FUNCTION_BLOCK CentralServerConveyorCTL (* Basic Function Block Type *)
  (* Standard: 61499-2 *)
  (* Version 0.2, 2003-12-04, JHC, Rockwell Automation, Renamed for better indexing. *)
  (* Version 0.1, 2002-11-05, JHC, Rockwell Automation, Corrected missing ST element in Algorithm REQ. *)
  (* Version 0.0, 2000-05-30, JHC, Rockwell Automation *)
  (* Compiler header: package fb.rt.cs725; *)
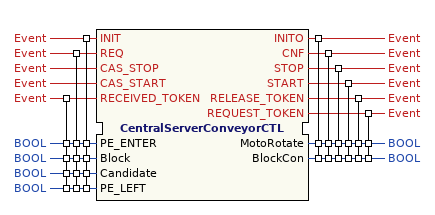
  EVENT_INPUT
    INIT WITH PE_ENTER, Block, Candidate, PE_LEFT; (* Initialization Request *)
    REQ WITH PE_ENTER, Block, Candidate, PE_LEFT; (* Normal Execution Request *)
    CAS_STOP;
    CAS_START;
    RECEIVED_TOKEN WITH PE_ENTER, Block, Candidate, PE_LEFT;
  END_EVENT
  EVENT_OUTPUT
    INITO WITH MotoRotate, BlockCon; (* Initialization Confirm *)
    CNF WITH MotoRotate, BlockCon; (* Execution Confirmation *)
    STOP WITH MotoRotate, BlockCon;
    START WITH BlockCon, MotoRotate;
    RELEASE_TOKEN WITH MotoRotate, BlockCon;
    REQUEST_TOKEN WITH MotoRotate, BlockCon;
  END_EVENT
  VAR_INPUT
    PE_ENTER : BOOL; (* Input event qualifier *)
    Block : BOOL;
    Candidate : BOOL;
    PE_LEFT : BOOL;
  END_VAR
  VAR_OUTPUT
    MotoRotate : BOOL; (* Output event qualifier *)
    BlockCon : BOOL;
  END_VAR
  VAR
    lastPE : BOOL := 1;
    lastBlock : BOOL := 0;
  END_VAR
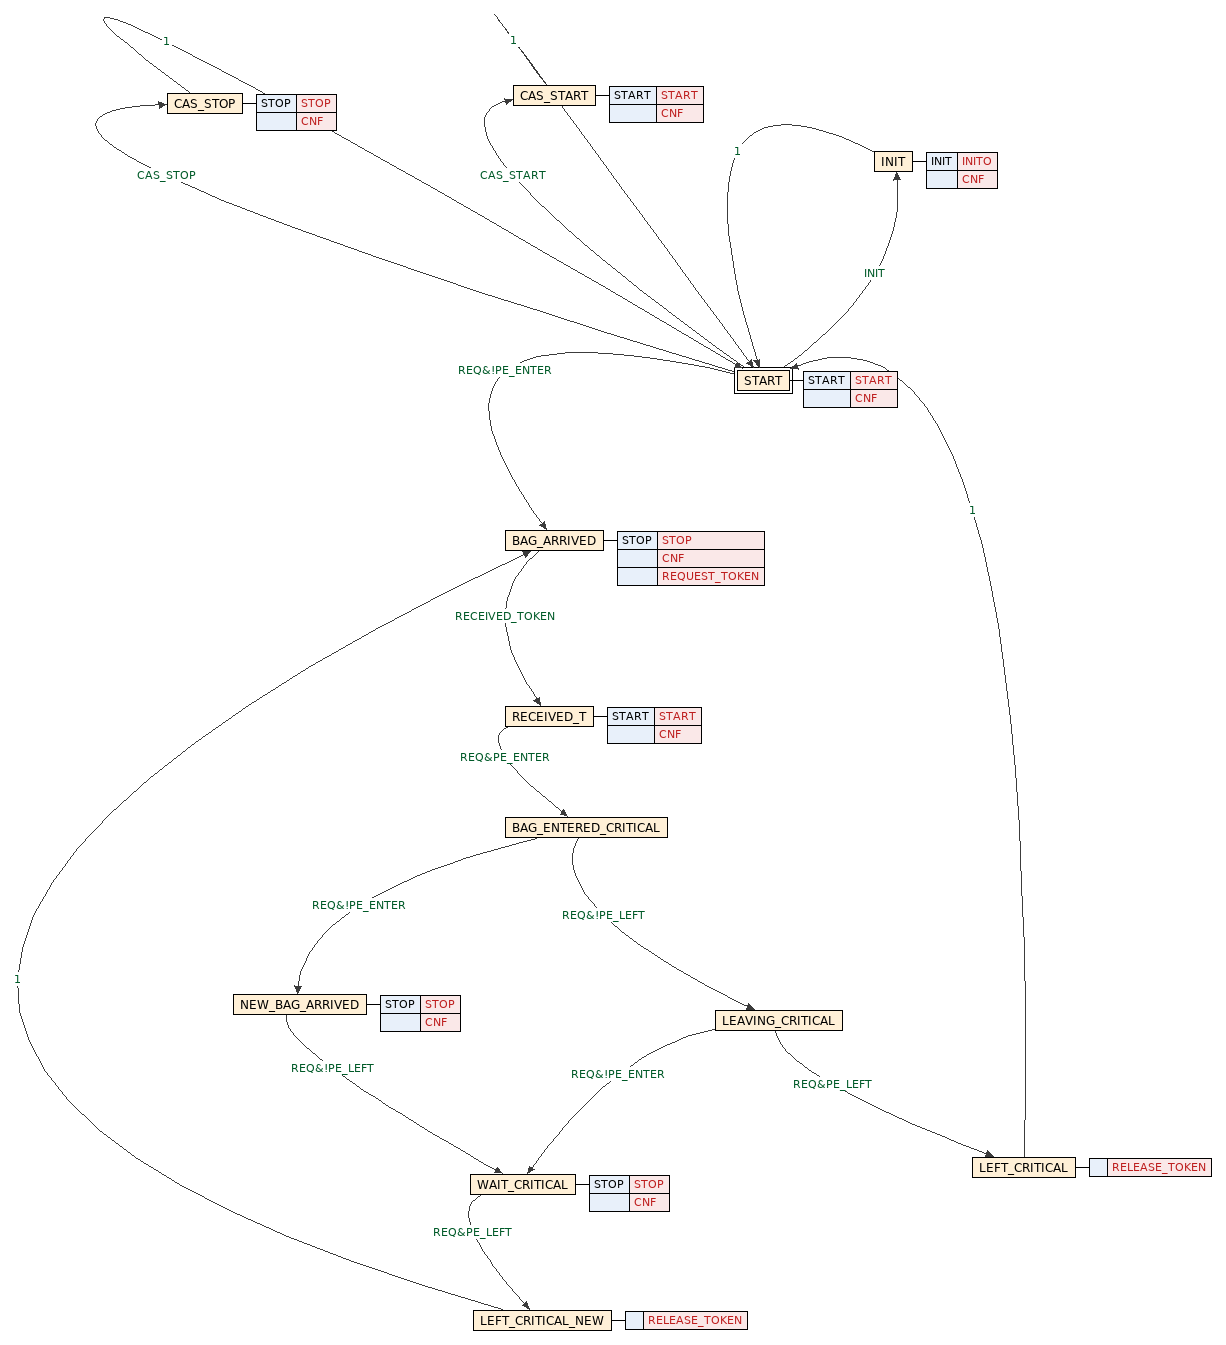
  EC_STATES
    START : START -> START, -> CNF; (* Initial State *)
    INIT : INIT -> INITO, -> CNF; (* Initialization *)
    BAG_ARRIVED : STOP -> STOP, -> CNF, -> REQUEST_TOKEN; (* Normal execution *)
    CAS_START : START -> START, -> CNF;
    CAS_STOP : STOP -> STOP, -> CNF;
    RECEIVED_T : START -> START, -> CNF; (* Token recived *)
    BAG_ENTERED_CRITICAL;
    NEW_BAG_ARRIVED : STOP -> STOP, -> CNF;
    LEAVING_CRITICAL;
    WAIT_CRITICAL : STOP -> STOP, -> CNF;
    LEFT_CRITICAL_NEW : -> RELEASE_TOKEN;
    LEFT_CRITICAL : -> RELEASE_TOKEN;
  END_STATES
  EC_TRANSITIONS
    START TO INIT := INIT;
    INIT TO START := 1;
    START TO BAG_ARRIVED := REQ&!PE_ENTER;
    START TO CAS_START := CAS_START;
    CAS_START TO START := 1;
    START TO CAS_STOP := CAS_STOP;
    CAS_STOP TO START := 1;
    BAG_ARRIVED TO RECEIVED_T := RECEIVED_TOKEN;
    RECEIVED_T TO BAG_ENTERED_CRITICAL := REQ&PE_ENTER;
    BAG_ENTERED_CRITICAL TO NEW_BAG_ARRIVED := REQ&!PE_ENTER;
    BAG_ENTERED_CRITICAL TO LEAVING_CRITICAL := REQ&!PE_LEFT;
    NEW_BAG_ARRIVED TO WAIT_CRITICAL := REQ&!PE_LEFT;
    LEAVING_CRITICAL TO WAIT_CRITICAL := REQ&!PE_ENTER;
    WAIT_CRITICAL TO LEFT_CRITICAL_NEW := REQ&PE_LEFT;
    LEFT_CRITICAL_NEW TO BAG_ARRIVED := 1;
    LEAVING_CRITICAL TO LEFT_CRITICAL := REQ&PE_LEFT;
    LEFT_CRITICAL TO START := 1;
  END_TRANSITIONS
  ALGORITHM INIT IN ST: (* Initialization algorithm *)
MotoRotate := TRUE;
Block := FALSE;

System.out.println(this + " " + MotoRotate);
System.out.println(MotoRotate);
  END_ALGORITHM
  ALGORITHM REQ IN ST: (* Normally executed algorithm *)
System.out.println(this +  " -> Candidate" + Candidate);
IF Candidate THEN
IF lastPE !:= PE_ENTER THEN
IF NOT PE_ENTER THEN
BlockCon:= TRUE;
System.out.println("BlockCon = true");
ELSE
BlockCon:=FALSE;
System.out.println("BlockCon = false");
END_IF
lastPE := PE_ENTER;
END_IF
IF lastBlock !:= Block THEN
IF Block THEN
STOP.serviceEvent(this);
MotoRotate := FALSE;
System.out.println("Cas Stop");
ELSE
START.serviceEvent(this);
MotoRotate := TRUE;
System.out.println("Cas Start");
END_IF
lastBlock := Block;
END_IF
END_IF
  END_ALGORITHM
  ALGORITHM START IN ST:
MotoRotate:=TRUE;
System.out.println(this + " Start " + MotoRotate);

System.out.println("Start " + MotoRotate);
  END_ALGORITHM
  ALGORITHM STOP IN ST:
MotoRotate := FALSE;
System.out.println(this + " Stop " + MotoRotate);

System.out.println("Stop " + MotoRotate);
  END_ALGORITHM
END_FUNCTION_BLOCK
